(* PLC project  *)

CONFIGURATION Empty_Module_18
END_CONFIGURATION
